{attribute 'TcGenerated'}
{attribute 'no-analysis'}
{attribute 'linkalways'}
// This function has been automatically generated from the project information.
VAR_GLOBAL CONSTANT
	{attribute 'const_non_replaced'}
	stLibVersion_TwinCAT_Dynamic_String_Kit : ST_LibVersion := (iMajor := 1, iMinor := 0, iBuild := 2, iRevision := 2, nFlags := 0, sVersion := '1.0.2.2');
END_VAR

(* stored: Version 1.1.0.1, ProductVersion 3.1.4024.4
   GVL Global_Version: Id {41ad341d-f938-4f02-8361-d54b5f714789} *)
